FUNCTION_BLOCK Infeed EXTENDS FB_PackML_BaseModule
VAR
	iInfeedxis				   : I_BasicAxis;				  // For most axis and component commands
	iInfeedAxisComponent	   : I_ComponentBase;			  // For registering the component with the EM
	iExternalSetpointGenerator : I_ExternalSetpointGenerator; // For setting properties of the External Setpoint Generator
END_VAR

// This method contains code which will execute when this PackML module is in the Aborting state
METHOD PROTECTED Aborting
VAR
	i				: UDINT;
	SubModulesReady : BOOL := TRUE;
END_VAR

// Note: The Abort command should be associated with the fault handing routine of a module. It should not be directly commanded from any user inteface. 

// This method is called as required by <c>StateControl()</c>
CASE SequenceState OF
	0:
		NoStateTasksToComplete := FALSE;
		SequenceState		   := SequenceState + 10;

	10:
		IF NOT iInfeedxis.Error THEN
			IF iInfeedxis.Stop() THEN
				SequenceState := SequenceState + 10;
			END_IF
		ELSE
			SequenceState := SequenceState + 10;
		END_IF

	20:
		IF iInfeedxis.Stopped THEN
			SequenceState := SequenceState + 10;
		END_IF

	30:
		IF iInfeedxis.Disable() THEN
			SequenceState := SequenceState + 10;
		END_IF

	40:
		IF NOT iInfeedxis.Enabled THEN
			SequenceState := SequenceState + 10;
		END_IF

	50:
		StateTasksComplete := TRUE;
END_CASE

SUPER^.Aborting();
END_METHOD

// This method contains code which will execute when this PackML module is in the Clearing state
METHOD PROTECTED Clearing
VAR
	i				: UDINT;
	SubModulesReady : BOOL := TRUE;
END_VAR

// Note: The Clear command can also be thought of as a fault reset depite the ambiguity in the naming of the Reset state. 

// This method is called as required by <c>StateControl()</c>
CASE SequenceState OF
	0:
		NoStateTasksToComplete := FALSE;
		SequenceState		   := SequenceState + 10;

	10:
		IF iInfeedxis.Reset() THEN
			SequenceState := SequenceState + 10;
		END_IF

	20:
		IF NOT iInfeedxis.Error THEN
			SequenceState := SequenceState + 10;
		END_IF

	30:
		StateTasksComplete := TRUE;
END_CASE

SUPER^.Clearing();
END_METHOD

// This method contains code which will execute when this PackML module is in the Execute state
METHOD PROTECTED Execute

(*
The base implementation of this method is empty. User must override this method to provide functionality.
This method is called as required by StateControl()
*)

VAR
	Position: LREAL;
END_VAR
CASE _CurrentMode OF
	E_PMLUnitMode.ePMLUnitMode_Production:
		CASE SequenceState OF
			0:
				iExternalSetpointGenerator.Direction   := 1;
				iExternalSetpointGenerator.Destination := 100.0;
				iExternalSetpointGenerator.Velocity	   := 0.0;
				iExternalSetpointGenerator.Accel	   := 0.0;
				SequenceState						   := 10;

			10:
				IF iInfeedxis.RunExternalSequence() THEN
					SequenceState := 20;
				END_IF

			20:
				IF iInfeedxis.Axis.Status.HasJob THEN //Setpoint generator is operational
					SequenceState := 30;
				END_IF

			30: // Move from 0 to Destination
				Position := iInfeedxis.ActualPosition + ((iExternalSetpointGenerator.Destination - iInfeedxis.ActualPosition) * 0.01);

				iExternalSetpointGenerator.Position := Position;
				IF iInfeedxis.InPosition THEN
					SequenceState := 40;
				END_IF

			40:
				IF iExternalSetpointGenerator.Disable() THEN
					SequenceState := 50;
				END_IF

			50:
				;
		END_CASE
END_CASE
END_METHOD

// Basic module initialization logic
METHOD PROTECTED Initialize : BOOL;
VAR
END_VAR

// This method is called by CyclicLogic() as required
Initialize := FALSE;
CASE DescendantSequenceState OF
	0:
		// Interfaces to connect to Components in the Fast_Task
		iInfeedxis				   := Fast_Task.PositionAxis;	   // For most axis and component commands
		iInfeedAxisComponent	   := Fast_Task.PositionAxis;	   // For registering the component with the EM
		iExternalSetpointGenerator := Fast_Task.PosExtSetpointGen; // For setting properties of the External Setpoint Generator

		//
		RegisterComponent(Component := iInfeedAxisComponent);
		DescendantSequenceState := DescendantSequenceState + 10;

	10:
		IF SUPER^.Initialize() THEN
			DescendantSequenceState := DescendantSequenceState + 10;
		END_IF

	20:
		Initialize := TRUE;
END_CASE
END_METHOD

METHOD PROTECTED Resetting
VAR
END_VAR
CASE SequenceState OF
	0:
		NoStateTasksToComplete := FALSE;
		SequenceState		   := SequenceState + 10;

	10:
		IF iInfeedxis.Enable() THEN
			SequenceState := SequenceState + 10;
		END_IF

	20:
		IF iInfeedxis.Enabled THEN
			SequenceState := SequenceState + 10;
		END_IF

	30:
		StateTasksComplete := TRUE;
END_CASE

SUPER^.Resetting();
END_METHOD

END_FUNCTION_BLOCK

(* stored: Version 1.1.0.1, ProductVersion 3.1.4024.12
   POU Infeed: Id {0bcf2b52-7ec2-4292-b061-d82e0eb4dd73}, SpecialFunc None
   Method Aborting: Id {22e9bc00-c001-4792-8e0c-9e46bc3906e9}
   Method Clearing: Id {3b500a04-f47d-487a-b737-898d3c9f4cfd}
   Method Execute: Id {4883edbf-5676-44d4-88e6-18721f181889}
   Method Initialize: Id {a90989da-9185-4daa-bb74-7f6195b68e99}
   Method Resetting: Id {3d1b53cb-4fac-4d3d-9bee-04f00ee33a88} *)
